FUNCTION SetBit : ULINT
VAR_INPUT
	Value: ULINT;
	BitNr: INT;
	State: BOOL;
END_VAR
VAR
END_VAR

IF State THEN
	SetBit := (Value AND (NOT SHL(INT_TO_ULINT(1), BitNr))) OR SHL(INT_TO_ULINT(1), BitNr);
ELSE
	SetBit := (Value AND (NOT SHL(INT_TO_ULINT(1), BitNr)));
END_IF

END_FUNCTION

(* stored: Version 1.1.0.1, ProductVersion 3.1.4024.3
   POU SetBit: Id {69b065bc-58cc-4bb0-8793-a161fe34eb32}, SpecialFunc None *)
